{attribute 'qualified_only'}
{attribute 'strict'}
TYPE E_PneumaticMode :
(   eSingleSolenoidControl := 0, //Single solenoid valve with spring return
    eReset := 1,
    eError := 2
):= eSingleSolenoidControl;
END_TYPE

(* stored: Version 1.1.0.1, ProductVersion 3.1.4024.12
   DUT E_PneumaticMode: Id {767ff514-f7ef-4e71-a359-d55b64a86d25} *)
